PROGRAM MAIN

HMI();
SDO();
STATE_MACHINE();

END_PROGRAM

(* stored: Version 1.1.0.1, ProductVersion 3.1.4024.11
   POU MAIN: Id {ee9132d2-9909-442e-a723-ffe0f98e05bb}, SpecialFunc None *)
